TYPE TestStruct :
STRUCT
	iVal : DINT := 0;
	fVal : REAL := 0.0;
	sVal : STRING := '';
END_STRUCT
END_TYPE

(* stored: Version 1.1.0.1, ProductVersion 3.1.4024.3
   DUT TestStruct: Id {945d4d07-6e76-44ab-9627-aa805f40351f} *)
